{attribute addProperty BoxType "AT2020-0250-0023"}
{attribute addProperty Id "A_0073_AT2000_5250_0016_AT2000_5250AT2000_C5E5984862678.25"}
{attribute addProperty CRC "254730196"}
{attribute addProperty SizeInBites "626"}
{attribute addProperty SizeInBytes "78.25"}
TYPE A_0061_AT2020_0250_0023_AT2020_0250_0F2EDFD4 EXTENDS AT2020_BA5A9548 :
STRUCT
	{attribute addProperty Name "A_0073_AT2000_5250_0016_AT2000_5250"}
	A_0073_AT2000_5250_0016_AT2000_5250 : AT2000_C5E59848;
END_STRUCT
END_TYPE

(* stored: Version 1.2.0.0, ProductVersion 3.1.4024.9
   DUT A_0061_AT2020_0250_0023_AT2020_0250_0F2EDFD4: Id {2419b50f-4536-4763-96df-6bdcdd870157} *)
